Staubli VAL3: pwrOffDrive2.pgx

public program pwrOffDrive2(num x_nAxNum)
  local bool l_bOK
  local string l_sMsg
begin
  // sequenceur pour desactiver les variateurs

  // Read current drive State
  call chkDrvState(x_nAxNum)

  // Changement d'état ?
  if nDrvState[x_nAxNum]!=nMemPwrOffStep[x_nAxNum]
    nMemPwrOffStep[x_nAxNum]=nDrvState[x_nAxNum]
    bLockPwrOff[x_nAxNum]=false
  endIf

  l_sMsg="pwrOffDrive>>Etape : "+toString("",nDrvState[x_nAxNum])+" "
  switch nDrvState[x_nAxNum]
    // Not ready to Switch on
    case 1
      if bLockPwrOff[x_nAxNum]==false
        if bAnd(nDebug,cst:nDEBUGDRIVE)==cst:nDEBUGDRIVE
          l_sMsg=l_sMsg+"Not ready to Switch on"
          logMsg(l_sMsg)
        endIf
        bLockPwrOff[x_nAxNum]=true
      endIf
    break
    // Switch ON disabled
    case 2
      if bLockPwrOff[x_nAxNum]==false
        if bAnd(nDebug,cst:nDEBUGDRIVE)==cst:nDEBUGDRIVE
          l_sMsg=l_sMsg+"Switch on disabled"
          logMsg(l_sMsg)
        endIf
        call cmdResetAll(x_nAxNum)
        bLockPwrOff[x_nAxNum]=true
      endIf
    break
    // Ready to switch on
    case 3
      if bLockPwrOff[x_nAxNum]==false
        if bAnd(nDebug,cst:nDEBUGDRIVE)==cst:nDEBUGDRIVE
          l_sMsg=l_sMsg+"Ready to switch on"
          logMsg(l_sMsg)
        endIf
        call cmdQuickStop(x_nAxNum)
        call cmdDisableVolt(x_nAxNum)
        bLockPwrOff[x_nAxNum]=true
      endIf
    break
    // Switched ON
    case 4
      if bLockPwrOff[x_nAxNum]==false
        if bAnd(nDebug,cst:nDEBUGDRIVE)==cst:nDEBUGDRIVE
          l_sMsg=l_sMsg+"Switched ON"
          logMsg(l_sMsg)
        endIf
        call cmdShutdown(x_nAxNum)
        bLockPwrOff[x_nAxNum]=true
      endIf
    break
    // Operation enabled
    case 5
      if bLockPwrOff[x_nAxNum]==false
        if bAnd(nDebug,cst:nDEBUGDRIVE)==cst:nDEBUGDRIVE
          l_sMsg=l_sMsg+"Operation enabled"
          logMsg(l_sMsg)
        endIf
        call cmdDisableOp(x_nAxNum)
        bLockPwrOff[x_nAxNum]=true
      endIf
    break

    // Fault state
    case 14
      if bLockPwrOff[x_nAxNum]==false
        if bAnd(nDebug,cst:nDEBUGDRIVE)==cst:nDEBUGDRIVE
          l_sMsg=l_sMsg+"Fault state"
          logMsg(l_sMsg)
        endIf
        bLockPwrOff[x_nAxNum]=true
      endIf
    break
    //
    // Alarm from status_remote register is set
    case 15
      if bLockPwrOff[x_nAxNum]==false
        if bAnd(nDebug,cst:nDEBUGDRIVE)==cst:nDEBUGDRIVE
          l_sMsg=l_sMsg+"Alarm Status_remote register"
          logMsg(l_sMsg)
        endIf
        call cmdResetAll(x_nAxNum)
        bLockPwrOff[x_nAxNum]=true
      endIf
    break
    //
  endSwitch

end
